Staubli VAL3: buildList.pgx

program buildList()
  local num l_nSize
  local string l_sEvent
  local num i
  local string l_sString
begin
  // INIT the list
  l_sString=""
  call use:stringCopy(l_sString,sList)
  // Build the list
  call axis:getSize(l_nSize)
  // check the list empty
  call axis:get(l_sEvent,0)
  if l_sEvent!=""
    for i=0 to (l_nSize-1)
      call axis:get(l_sEvent,i)
      if l_sEvent!=""
        call listAdd(toString("2",i+1)+" "+l_sEvent)
      endIf
    endFor
  endIf

end
